# EPICS autosave request: ipApp/Db/PTC10_tc_chan_settings.req
$(P)$(T):$(C):temperature.SCAN
#$(P)$(T):$(C):sensor
